Staubli VAL3: set.pgx

public program set(string x_sName, string x_sItem)
begin
  // Get IT
  //  sName[x_nIndex]=x_sItem
  if isDefined(saveInOut:cCount[x_sItem])
    saveInOut:cCount[x_sItem].sName=x_sName
  elseIf isDefined(saveInOut:aCount[x_sItem])
    saveInOut:aCount[x_sItem].sName=x_sName
  else
    // not found
    // toDO
    popUpMsg("value not found: "+x_sItem)
    x_sItem=""
  endIf
end
